///EL2902 | 2-channel digital output terminal, TwinSAFE, 24 V DC, 2.3 A
FUNCTION_BLOCK EL2902_v0_00

END_FUNCTION_BLOCK

(* stored: Version 1.1.0.1, ProductVersion 3.1.4022.6
   POU EL2902_v0_00: Id {780e7f23-9c93-465a-8965-e5bf0ecffc55}, SpecialFunc None *)
